short summary
=================
This methode returns the next object in the iteration and returns an execution state.
Example:
You have a list: 1 2 3
the first iterate call will return CNM_ReturnTypes.BUSY and object = 1
the second iterate call will return CNM_ReturnTypes.BUSY and object = 2
the third iterate call will return CNM_ReturnTypes.SUCCESS and object = 3

.. <legal notes>

legal notes
=================
| SPDX-FileCopyrightText: © 2022 ekvip automation GmbH <info@ekvip.de>
| SPDX-License-Identifier: Apache-2.0
| For details check: Apache-2.0_

.. _Apache-2.0: https://www.apache.org/licenses/LICENSE-2.0

.. </legal notes>

parameters
=================

*)
METHOD iterate : CNM_ReturnTypes.SingleExecutionState
VAR_INPUT
	(*control bit to start or abort the iterate*)
	execute	: BOOL;
END_VAR
VAR_OUTPUT
	(*the returned object of the iteration*)
	line	: ILine;
END_VAR
VAR
	tmp : IObject;
END_VAR
iterate := THIS^.list.iterate(execute := execute, object => tmp);
__QUERYINTERFACE(tmp, line);
END_METHOD

(*

short summary
=================
This property returns the last object in the list and removes it from the list. Can be seen as opposite of append.
Example:
On a list: (Head -->) A B C, list.pop will return C.
Example 2:
If you call append(x), a pop right after will return x.
May return a null pointer if list is empty

.. <legal notes>

legal notes
=================
| SPDX-FileCopyrightText: © 2022 ekvip automation GmbH <info@ekvip.de>
| SPDX-License-Identifier: Apache-2.0
| For details check: Apache-2.0_

.. _Apache-2.0: https://www.apache.org/licenses/LICENSE-2.0

.. </legal notes>

*)
METHOD pop : ILine
__QUERYINTERFACE(THIS^.list.pop(), pop);
END_METHOD

(*

short summary
=================
This methode adds the given obejct to the end of the list.
Example: 
Given a list that looks like this: (Head->) A B C (<- End),
calling prepend(D) on this list will place the D at start,
making it the new Head: (Head->) D A B C (<- End)

.. <legal notes>

legal notes
=================
| SPDX-FileCopyrightText: © 2022 ekvip automation GmbH <info@ekvip.de>
| SPDX-License-Identifier: Apache-2.0
| For details check: Apache-2.0_

.. _Apache-2.0: https://www.apache.org/licenses/LICENSE-2.0

.. </legal notes>

parameters
=================
:return: ``SingleExecutionResult.SUCCESS``: prepend was successful
	``SingleExecutionResult.ERROR``: allocation of memory for new object failed
	
*)
METHOD prepend : CNM_ReturnTypes.SingleExecutionResult
VAR_INPUT
	(*The object to be prepended*)
	line	: ILine;
END_VAR
prepend := THIS^.list.prepend(object := line);
END_METHOD

(*

short summary
=================
This methode adds all elements of the given collection to the start of this list. 
Example:
For the list1: A B C and list2: D E F will be after list1.prependCollection(list2):
D E F A B C. Notice the elements are still in the same order they where befor on each subsection.

.. <legal notes>

legal notes
=================
| SPDX-FileCopyrightText: © 2022 ekvip automation GmbH <info@ekvip.de>
| SPDX-License-Identifier: Apache-2.0
| For details check: Apache-2.0_

.. _Apache-2.0: https://www.apache.org/licenses/LICENSE-2.0

.. </legal notes>

parameters
=================
:return: ``SingleExecutionResult.SUCCESS``: prependCollection was successful
	``SingleExecutionResult.ERROR``: could not allocate memory for all new elements, list is left unchanged

*)
METHOD prependCollection : CNM_ReturnTypes.SingleExecutionResult
VAR_INPUT
	(*The collection to be prepended*)
	collectionToPrepend	: CNM_CollectionInterfaces.ICollection;
END_VAR
prependCollection := THIS^.list.prependCollection(collectionToPrepend := collectionToPrepend);
END_METHOD

(*

short summary
=================
This methode removes the first instance of the given object from the list.
Compares objects with hash value.
For example a Linked List: A B C A A D will on remove(A) becomes: B C A A D

.. <legal notes>

legal notes
=================
| SPDX-FileCopyrightText: © 2022 ekvip automation GmbH <info@ekvip.de>
| SPDX-License-Identifier: Apache-2.0
| For details check: Apache-2.0_

.. _Apache-2.0: https://www.apache.org/licenses/LICENSE-2.0

.. </legal notes>

parameters
=================

*)
METHOD remove
VAR_INPUT
	(*The object to be removed from the list*)
	line	: ILine;
END_VAR
THIS^.list.remove(object := line);
END_METHOD

(*

short summary
=================
This methode removes the element at the given index. 
Will shift the remaining data to the left (no empty space in list)
List Length will be decremented.
Example:
A list of: 1 2 3 after list.removeObjectAt(1) will become: 1 3 and return IndexBounds.IN_BOUNDS
Example 2:
A list of: 1 2 3 after list.removeObjectAt(3) will reamin: 1 2 3 and return IndexBounds.OUT_OF_BOUNDS

.. <legal notes>

legal notes
=================
| SPDX-FileCopyrightText: © 2022 ekvip automation GmbH <info@ekvip.de>
| SPDX-License-Identifier: Apache-2.0
| For details check: Apache-2.0_

.. _Apache-2.0: https://www.apache.org/licenses/LICENSE-2.0

.. </legal notes>

parameters
=================
:return: ``SingleExecutionResult.SUCCESS``: Element removed from index
    ``SingleExecutionResult.ERROR``: index out of bound, no object removed

*)
METHOD removeLineAt : CNM_ReturnTypes.SingleExecutionResult
VAR_INPUT
	(*the index to remove the object from*)
	index	: __XWORD;
END_VAR
removeLineAt := THIS^.list.removeObjectAt(index := index);
END_METHOD

(*

short summary
=================
This methode replaces the Interface reference inside the collection at the given index with the given Interface.
Example:
A list of: 1 2 3 after list.replaceObjectAt(1, withObject:=4) will become: 1 4 3 and return SingleExecutionResult.SUCCESS
Example 2:
A list of: 1 2 3 after list.replaceObjectAt(3, withObject:=4) will remain: 1 2 3 and return SingleExecutionResult.ERROR

.. <legal notes>

legal notes
=================
| SPDX-FileCopyrightText: © 2022 ekvip automation GmbH <info@ekvip.de>
| SPDX-License-Identifier: Apache-2.0
| For details check: Apache-2.0_

.. _Apache-2.0: https://www.apache.org/licenses/LICENSE-2.0

.. </legal notes>

parameters
=================
:return: ``SingleExecutionResult.SUCCESS``: index valid, element at index replaced with ``withObject``
    ``SingleExecutionResult.ERROR``: ìndex out of bounds, nothing changed

*)
METHOD replaceLineAt : CNM_ReturnTypes.SingleExecutionResult
VAR_INPUT
	(*the index to replace the object at*)
	index	: __XWORD;
	(*the object to be at this index instead*)
	withLine	: ILine;
END_VAR
replaceLineAt := THIS^.list.replaceObjectAt(index := index, withObject := withLine);
END_METHOD

(*

short summary
=================
This methode can replace the default sorter for a custom one. Check :ref:`IListSorter`
Can be used for performant sorting algorithms if more about the data structure is known.

.. attention:: 
	For implementations: **IListSorter is an empty interface and you should extend it with custom interfaces for each type of list.**
	For LinkedList see :ref:`ILinkedListSorter`. 
	Your implementation should then use this extended interface and the setter should check for compability. 
	
.. <legal notes>

legal notes
=================
| SPDX-FileCopyrightText: © 2022 ekvip automation GmbH <info@ekvip.de>
| SPDX-License-Identifier: Apache-2.0
| For details check: Apache-2.0_

.. _Apache-2.0: https://www.apache.org/licenses/LICENSE-2.0

.. </legal notes>

parameters
=================
:return: ``THIS^`` :ref:`IList`

*)
METHOD setSorter : CNM_CollectionInterfaces.ISortable
VAR_INPUT
	(*The instance of the sorter to be used to sort the list*)
	sorter	: CNM_CollectionInterfaces.IArrayListSorter;
END_VAR
setSorter := THIS^.list.setSorter(sorter := sorter);
END_METHOD

(*

short summary
=================
This property returns the number of elements inside this collection.

.. <legal notes>

legal notes
=================
| SPDX-FileCopyrightText: © 2022 ekvip automation GmbH <info@ekvip.de>
| SPDX-License-Identifier: Apache-2.0
| For details check: Apache-2.0_

.. _Apache-2.0: https://www.apache.org/licenses/LICENSE-2.0

.. </legal notes>

*)
PROPERTY size : __XWORD
GET
size := THIS^.list.size;
END_GET
END_PROPERTY

(*

short summary
=================
This method sorts the data structure. 
This can take many cycles and should be called until the CNM_ReturnTypes.ExecutionState is no longer ``BUSY``.

.. <legal notes>

legal notes
=================
| SPDX-FileCopyrightText: © 2022 ekvip automation GmbH <info@ekvip.de>
| SPDX-License-Identifier: Apache-2.0
| For details check: Apache-2.0_

.. _Apache-2.0: https://www.apache.org/licenses/LICENSE-2.0

.. </legal notes>

parameters
=================
:return: ``ABORTED``: While sort was pending,execute had a falling edge,
	``BUSY``: Sort is in progress
	``ERROR``: Sort was not able to finish (p.e. List changed) call sort(false) to reset
	``IDLE``: Currently no sort in progress
	``SUCCESS``: Sorting was finished 

*)
METHOD sort : CNM_ReturnTypes.SingleExecutionState
VAR_INPUT
	(*control bit to start or abort the sorting, needs to be active until the ExecutionState is SUCCESS*)
	execute	: BOOL;
END_VAR
sort := THIS^.list.sort(execute := execute);
END_METHOD

(*

short summary
=================
This method sorts the data structure. 
It uses the passed Comperator to sort the structure.
This can take many cycles and should be called until the CNM_ReturnTypes.ExecutionState is no longer ``BUSY``.

.. <legal notes>

legal notes
=================
| SPDX-FileCopyrightText: © 2022 ekvip automation GmbH <info@ekvip.de>
| SPDX-License-Identifier: Apache-2.0
| For details check: Apache-2.0_

.. _Apache-2.0: https://www.apache.org/licenses/LICENSE-2.0

.. </legal notes>

parameters
=================
:return: ``ABORTED``: While sort was pending,execute had a falling edge,
	``BUSY``: Sort is in progress
	``ERROR``: Sort was not able to finish (p.e. List changed) call sort(false) to reset
	``IDLE``: Currently no sort in progress
	``SUCCESS``: Sorting was finished 

*)
METHOD sortWithComparator : CNM_ReturnTypes.SingleExecutionState
VAR_INPUT
	(*control bit to start or abort the sorting, needs to be active until the ExecutionState is SUCCESS*)
	execute	: BOOL;
	(*the comparator that should be used for the sort. Must not be changed while sort is in process*)
	comparator	: CNM_AbstractObject.IComparator;
END_VAR
sortWithComparator := THIS^.list.sortWithComparator(execute := execute, comparator := comparator);
END_METHOD

END_FUNCTION_BLOCK

// ---- Value/UlintValue.TcPOU
FUNCTION_BLOCK UlintValue EXTENDS Object IMPLEMENTS IHaveUlintValue
VAR
	myValue :ULINT;
END_VAR

(*

short summary
=================
This abstract property returns the class name of the concrete object, 
which is useful for logging/debugging purpose or to check the class name
for ``__DELETE`` in factories (sometimes it's necessary to do more 
than just to free the memory).

.. <legal notes>

legal notes
=================
| SPDX-FileCopyrightText: © 2022 ekvip automation GmbH <info@ekvip.de>
| SPDX-License-Identifier: Apache-2.0
| For details check: Apache-2.0_

.. _Apache-2.0: https://www.apache.org/licenses/LICENSE-2.0

.. </legal notes>

*)
PROPERTY className : CNM_AbstractObject.ClassName
GET
END_GET
END_PROPERTY

(*

short summary
=================
This method compares a foreign object with the own one, this is needed for sort orders.
The abstract class evaluates every object that is NULL as greater, and all other objects as equal. 

.. attention:: 
	For derivations: **If a derived class needs sorting this method must be overwritten.** 

.. <legal notes>

legal notes
=================
| SPDX-FileCopyrightText: © 2022 ekvip automation GmbH <info@ekvip.de>
| SPDX-License-Identifier: Apache-2.0
| For details check: Apache-2.0_

.. _Apache-2.0: https://www.apache.org/licenses/LICENSE-2.0

.. </legal notes>

parameters
=================
:return:``SMALLER``: ``THIS`` precedes in order,
``EQUAL``: ``THIS`` and ``object`` at the same position in order,
``GREATER``: ``THIS`` is after in order.
Checkout the library CNM_ReturnTypes.

*)
METHOD compareTo : CNM_AbstractObject.CNM_ReturnTypes.ComparationResult
VAR_INPUT
	(* foreign objet to compare*)
	object	: CNM_AbstractObject.IObject;
END_VAR
VAR
	other :IHaveValue;
END_VAR
compareTo := CNM_ReturnTypes.ComparationResult.EQUAL;

RETURN (object = 0);

IF(__QUERYINTERFACE(object, other))THEN
	IF(THIS^.value > other.value)THEN
		compareTo := CNM_ReturnTypes.ComparationResult.GREATER;
	ELSIF(THIS^.value < other.value)THEN
		compareTo := CNM_ReturnTypes.ComparationResult.SMALLER;
	END_IF
END_IF
END_METHOD

{warning 'Add property implementation'}
PROPERTY value : ULINT
GET
value := myValue;
END_GET
SET
myValue := value;
END_SET
END_PROPERTY

END_FUNCTION_BLOCK

// ---- Value/ValueSum.TcPOU
FUNCTION_BLOCK ValueSum EXTENDS AbstractApplier
VAR
	valueObject :IHaveValue;
	mySum :LREAL;
END_VAR

(*

short summary
=================
Methode to accept an object.
Example:
NumberIncrementer.accept(Number);

.. <legal notes>

legal notes
=================
| SPDX-FileCopyrightText: © 2022 ekvip automation GmbH <info@ekvip.de>
| SPDX-License-Identifier: Apache-2.0
| For details check: Apache-2.0_

.. _Apache-2.0: https://www.apache.org/licenses/LICENSE-2.0

.. </legal notes>

parameters
=========================

*)
METHOD accept : CNM_CollectionInterfaces.CNM_ReturnTypes.SingleExecutionResult
VAR_INPUT
	(*object to accept*)
	object	: CNM_CollectionInterfaces.CNM_AbstractObject.IObject;
END_VAR
IF(__QUERYINTERFACE(object, THIS^.valueObject))THEN
	accept := CNM_ReturnTypes.SingleExecutionResult.SUCCESS;
ELSE
	accept := CNM_ReturnTypes.SingleExecutionResult.ERROR;
END_IF
END_METHOD

(*

short summary
=================
A method to apply the concrete action on the given object (THIS^.object)

.. <legal notes>

legal notes
=================
| SPDX-FileCopyrightText: © 2022 ekvip automation GmbH <info@ekvip.de>
| SPDX-License-Identifier: Apache-2.0
| For details check: Apache-2.0_

.. _Apache-2.0: https://www.apache.org/licenses/LICENSE-2.0

.. </legal notes>

parameters
=========================
:return: CNM_ReturnTypes.ExecutionState

*)
METHOD apply : CNM_CollectionInterfaces.CNM_ReturnTypes.SingleExecutionState
VAR_INPUT
	(*control bit to start or abort the application, should to be active until the ExecutionState is SUCCESS*)
	execute	: BOOL;
END_VAR
RETURN (NOT execute);

apply := CNM_ReturnTypes.SingleExecutionState.ERROR;

RETURN (THIS^.isObjectNull(THIS^.valueObject));

apply := CNM_ReturnTypes.SingleExecutionState.SUCCESS;
THIS^.sum := THIS^.sum + THIS^.valueObject.value;
END_METHOD

(*

short summary
=================
This abstract property returns the class name of the concrete object, 
which is useful for logging/debugging purpose or to check the class name
for ``__DELETE`` in factories (sometimes it's necessary to do more 
than just to free the memory).

.. <legal notes>

legal notes
=================
| SPDX-FileCopyrightText: © 2022 ekvip automation GmbH <info@ekvip.de>
| SPDX-License-Identifier: Apache-2.0
| For details check: Apache-2.0_

.. _Apache-2.0: https://www.apache.org/licenses/LICENSE-2.0

.. </legal notes>

*)
PROPERTY className : CNM_AbstractObject.ClassName
GET
className := 'AOC.ValueSum';
END_GET
END_PROPERTY

PROPERTY sum : LREAL
GET
sum := THIS^.mySum;
END_GET
SET
THIS^.mySum := sum;
END_SET
END_PROPERTY

END_FUNCTION_BLOCK

// ---- Value/LintValue.TcPOU
FUNCTION_BLOCK LintValue EXTENDS Object IMPLEMENTS IHaveLintValue
VAR
	myValue :LINT;
END_VAR

(*

short summary
=================
This abstract property returns the class name of the concrete object, 
which is useful for logging/debugging purpose or to check the class name
for ``__DELETE`` in factories (sometimes it's necessary to do more 
than just to free the memory).

.. <legal notes>

legal notes
=================
| SPDX-FileCopyrightText: © 2022 ekvip automation GmbH <info@ekvip.de>
| SPDX-License-Identifier: Apache-2.0
| For details check: Apache-2.0_

.. _Apache-2.0: https://www.apache.org/licenses/LICENSE-2.0

.. </legal notes>

*)
PROPERTY className : CNM_AbstractObject.ClassName
GET
END_GET
END_PROPERTY

(*

short summary
=================
This method compares a foreign object with the own one, this is needed for sort orders.
The abstract class evaluates every object that is NULL as greater, and all other objects as equal. 

.. attention:: 
	For derivations: **If a derived class needs sorting this method must be overwritten.** 

.. <legal notes>

legal notes
=================
| SPDX-FileCopyrightText: © 2022 ekvip automation GmbH <info@ekvip.de>
| SPDX-License-Identifier: Apache-2.0
| For details check: Apache-2.0_

.. _Apache-2.0: https://www.apache.org/licenses/LICENSE-2.0

.. </legal notes>

parameters
=================
:return:``SMALLER``: ``THIS`` precedes in order,
``EQUAL``: ``THIS`` and ``object`` at the same position in order,
``GREATER``: ``THIS`` is after in order.
Checkout the library CNM_ReturnTypes.

*)
METHOD compareTo : CNM_AbstractObject.CNM_ReturnTypes.ComparationResult
VAR_INPUT
	(* foreign objet to compare*)
	object	: CNM_AbstractObject.IObject;
END_VAR
VAR
	other :IHaveValue;
END_VAR
compareTo := CNM_ReturnTypes.ComparationResult.EQUAL;

RETURN (object = 0);

IF(__QUERYINTERFACE(object, other))THEN
	IF(THIS^.value > other.value)THEN
		compareTo := CNM_ReturnTypes.ComparationResult.GREATER;
	ELSIF(THIS^.value < other.value)THEN
		compareTo := CNM_ReturnTypes.ComparationResult.SMALLER;
	END_IF
END_IF
END_METHOD

{warning 'Add property implementation'}
PROPERTY value : LINT
GET
value := myValue;
END_GET
SET
myValue := value;
END_SET
END_PROPERTY

END_FUNCTION_BLOCK
